TYPE ST_XZ_Point :
STRUCT
	X,
	Z : LREAL;
END_STRUCT
END_TYPE

(* stored: Version 1.1.0.1
   DUT ST_XZ_Point: Id {3ffc9b83-c943-4dfb-a9fd-ce0a8e76f9a3} *)
